{attribute 'qualified_only'}
VAR_GLOBAL
END_VAR

(* stored: Version 1.1.0.1, ProductVersion 3.1.4024.9
   GVL SystemVariables: Id {8cc71902-54f3-4068-b684-2ff92871ee93} *)
